// TIA Portal V21 export
TYPE "Std_Stazioni"
   STRUCT
      IN : Struct
         Possibile : Bool;
         Selezionato : Bool;
         Attivo : Bool;
      END_STRUCT;
      Prm : Struct
         BypassChiamata : Bool;   // Se impostato ad 1 la stazione chiama anche se la sua destinazione non è la momento in chiamata
      END_STRUCT;
   END_STRUCT;
END_TYPE
